(* Logix 5000 project; controller PRG_SIMON Emulate 5570 rev 30.12; software revision 30.00 *)

TASK MainTask (continuous, watchdog 5000 ms) : MainProgram

MODULES
   Local : Emulate 5570 (ICP 2, rev 30.12)
       : vendor 1 type 0 code 15 (ICP 0, rev 1.1, Output RPI 50 ms)
END_MODULES

TYPE UDT_BA :
STRUCT
   AL : BOOL[128];
END_STRUCT
END_TYPE

PROGRAM MainProgram   (* main routine MainRoutine *)
VAR
   PRG_Counter : DINT[2];
   PRG_i : DINT;
   PRG_j : DINT;
   PRG_Res_Len : DINT;
   PRG_Result : DINT[256];
   SCAN_CYCLE_TIME : DINT;
   Simon_Ciphertext : DINT[2,2];
   Simon_dec_i : DINT;
   Simon_dec_j : DINT;
   Simon_enc_i : DINT;
   Simon_enc_j : DINT;
   Simon_i : DINT;
   Simon_j : DINT;
   Simon_Plaintext : DINT[2,2];
   Simon_Rd_Max : DINT;
   Simon_Rotate_Result : DINT[2];
   Simon_Round_Keys : DINT[72,2];
   Simon_tmp1 : DINT[2];
   Simon_tmp2 : DINT[2];
   Simon_Ver : DINT;
   Simon_x : DINT[2];
   Simon_y : DINT[2];
END_VAR

ROUTINE MainRoutine   (* ladder *)
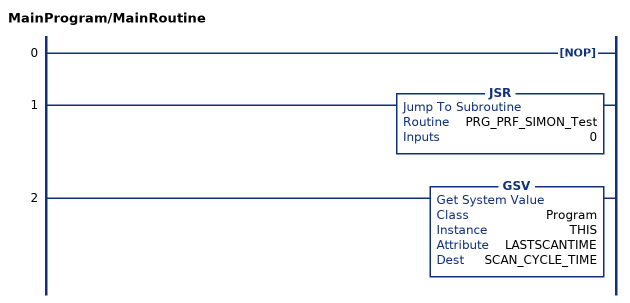
   0: NOP();
   1: JSR(PRG_PRF_SIMON_Test,0);
   2: GSV(Program,THIS,LASTSCANTIME,SCAN_CYCLE_TIME);
END_ROUTINE

ROUTINE PRG_PRF_Init   (* structured text *)
   
   
   //initialize version
   
   Simon_Ver:=2;     // 0: 32/64, 1: 64: 96, 2: 64:128, 3:128/128, 4:128/192, 5: 128/256
   
   PRG_j:=0;
   PRG_Res_Len :=  (PRG_Counter[0] AND 16#0000ffff)-1;
   
   JSR(SIMON_Init);
END_ROUTINE

ROUTINE PRG_PRF_SIMON   (* structured text *)
   // init PRG_Count[0] and PRG_Count[1] during application.. for PRF.. they could be any values
   //For PRG application, PRG_Count[0] defines the output length (i.e., the number of 64-bit, e.g., 128-bit output, PRG_Count[0]:=2)
   
   
   JSR(PRG_PRF_Init);
   PRG_j:=0;
   For PRG_i:=0 to PRG_Res_Len by 1 do
   	Simon_Plaintext[0,0]:=PRG_Counter[0]; //Upper bits of current plaintext
   	Simon_Plaintext[1,0]:=PRG_Counter[1];  //Lower bits of current plaintext
   	JSR(SIMON_Enc);
   	PRG_Result[PRG_j]:=Simon_Ciphertext[0,0];
   	PRG_Result[PRG_j+1]:=Simon_Ciphertext[1,0];
   
   	PRG_j:=PRG_j+2;
   
   End_For;
   
   JSR(SIMON_ClearKey);
   
END_ROUTINE

ROUTINE PRG_PRF_SIMON_Test   (* structured text *)
   If S:FS Then
   
   	PRG_Counter[0]:=5;
   	PRG_Counter[1]:=1;
   
   
   End_if;
   
   
   JSR(PRG_PRF_SIMON);
   
   
END_ROUTINE

ROUTINE SIMON_ClearKey   (* structured text *)
   Case Simon_Ver Of
   
   0,1,2:
   	For Simon_i:=0 to Simon_Rd_Max by 1 do
   		Simon_Round_Keys[Simon_i,0]:=0;
   	End_For;
   	Simon_tmp1[0]:=0;
   	Simon_tmp2[0]:=0;
   	Simon_Rotate_Result[0]:=0;
   3,4,5:
   	For Simon_i:=0 to Simon_Rd_Max by 1 do
   		Simon_Round_Keys[Simon_i,0]:=0;
   		Simon_Round_Keys[Simon_i,1]:=0;
   	End_For;
   	Simon_tmp1[0]:=0;
   	Simon_tmp1[1]:=0;
   	Simon_tmp2[0]:=0;
   	Simon_tmp2[1]:=0;
   	Simon_Rotate_Result[0]:=0;
   	Simon_Rotate_Result[1]:=0;
   End_Case;
   
   
END_ROUTINE

ROUTINE SIMON_Dec   (* structured text *)
   
   JSR(SIMON_Init);
   
   
   
   
   Case Simon_Ver Of
   
   0,1,2:
   	Simon_Plaintext[1,0]:=Simon_Ciphertext[0,0];
   	Simon_Plaintext[0,0]:=Simon_Ciphertext[1,0];
   
   	For Simon_i:=Simon_Rd_Max to 0 by -1 do
   		Simon_tmp2[0]:=Simon_Plaintext[0,0];  //for rotate
   		JSR(SIMON_Rotate_Left1);	//rotate based on Simon_Ciphertext[0,0]
   		Simon_tmp1[0]:= Simon_Rotate_Result[0];
   		Simon_Rotate_Result[0]:=0;
   
   		Simon_tmp2[0]:=Simon_Plaintext[0,0];  //for rotate
   		JSR(SIMON_Rotate_Left8);
   		Simon_tmp2[0]:=Simon_Rotate_Result[0];
   		Simon_tmp1[0]:= Simon_tmp1[0] AND Simon_tmp2[0];
   		Simon_Rotate_Result[0]:=0;
   
   		Simon_tmp2[0]:=Simon_Plaintext[0,0];  //for rotate
   		JSR(SIMON_Rotate_Left2);
   		Simon_tmp1[0]:= Simon_tmp1[0] XOR Simon_Rotate_Result[0];
   
   		Simon_tmp1[0]:= Simon_tmp1[0] XOR Simon_Round_Keys[Simon_i,0];
   
   		Simon_Plaintext[0,0]:= Simon_Plaintext[1,0] XOR Simon_tmp1[0];
   		Simon_Plaintext[1,0]:= Simon_tmp2[0];
   
   		Simon_Rotate_Result[0]:=0;
   
   	End_for;
   
   3,4,5:
   	Simon_Plaintext[1,0]:=Simon_Ciphertext[0,0];
   	Simon_Plaintext[1,1]:=Simon_Ciphertext[0,1];
   	Simon_Plaintext[0,0]:=Simon_Ciphertext[1,0];
   	Simon_Plaintext[0,1]:=Simon_Ciphertext[1,1];
   
   	For Simon_i:=Simon_Rd_Max to 0 by -1 do
   
   		Simon_tmp2[0]:=Simon_Plaintext[0,0];  //for rotate
   		Simon_tmp2[1]:=Simon_Plaintext[0,1];
   
   		JSR(SIMON_Rotate_Left1);	//rotate based on Simon_Ciphertext[0,0] and [0,1]
   		Simon_tmp1[0]:= Simon_Rotate_Result[0];
   		Simon_tmp1[1]:= Simon_Rotate_Result[1];
   
   		Simon_Rotate_Result[0]:=0;
   		Simon_Rotate_Result[1]:=0;
   
   		Simon_tmp2[0]:=Simon_Plaintext[0,0];
   		Simon_tmp2[1]:=Simon_Plaintext[0,1];
   		JSR(SIMON_Rotate_Left8);
   		Simon_tmp2[0]:=Simon_Rotate_Result[0];
   		Simon_tmp2[1]:=Simon_Rotate_Result[1];
   		Simon_tmp1[0]:= Simon_tmp1[0] AND Simon_tmp2[0];
   		Simon_tmp1[1]:= Simon_tmp1[1] AND Simon_tmp2[1];
   
   		Simon_tmp2[0]:=Simon_Plaintext[0,0];
   		Simon_tmp2[1]:=Simon_Plaintext[0,1];
   
   		Simon_Rotate_Result[0]:=0;
   		Simon_Rotate_Result[1]:=0;
   
   		JSR(SIMON_Rotate_Left2);
   		Simon_tmp1[0]:= Simon_tmp1[0] XOR Simon_Rotate_Result[0];
   		Simon_tmp1[1]:= Simon_tmp1[1] XOR Simon_Rotate_Result[1];
   
   		Simon_tmp1[0]:= Simon_tmp1[0] XOR Simon_Round_Keys[Simon_i,0];
   		Simon_tmp1[1]:= Simon_tmp1[1] XOR Simon_Round_Keys[Simon_i,1];
   
   
   		Simon_Plaintext[0,0]:= Simon_Plaintext[1,0] XOR Simon_tmp1[0];
   		Simon_Plaintext[0,1]:= Simon_Plaintext[1,1] XOR Simon_tmp1[1];
   
   		Simon_Plaintext[1,0]:= Simon_tmp2[0];
   		Simon_Plaintext[1,1]:= Simon_tmp2[1];
   
   		Simon_Rotate_Result[0]:=0;
   		Simon_Rotate_Result[1]:=0;
   
   	End_for;
   
   End_Case;
   
   
   
   
   
   
   JSR(SIMON_ClearKey);
   
   
   
   
   
   
   
   
END_ROUTINE

ROUTINE SIMON_Enc   (* structured text *)
   
   Case Simon_Ver Of
   
   0,1,2:
   	//Simon_Ciphertext[1,0]:=Simon_Plaintext[0,0];
   	//Simon_Ciphertext[0,0]:=Simon_Plaintext[1,0];
   
   	Simon_Ciphertext[0,0]:=Simon_Plaintext[1,0];
   	Simon_Ciphertext[1,0]:=Simon_Plaintext[0,0];
   
   	For Simon_i:=0 to Simon_Rd_Max by 1 do
   		Simon_tmp2[0]:=Simon_Ciphertext[0,0];  //for rotate
   		JSR(SIMON_Rotate_Left1);	//rotate based on Simon_Plaintext[0,0]
   		Simon_tmp1[0]:= Simon_Rotate_Result[0];
   		Simon_Rotate_Result[0]:=0;
   
   		Simon_tmp2[0]:=Simon_Ciphertext[0,0];  //for rotate
   		JSR(SIMON_Rotate_Left8);
   		Simon_tmp2[0]:=Simon_Rotate_Result[0];
   
   		Simon_tmp1[0]:= Simon_tmp1[0] AND Simon_tmp2[0];
   		Simon_Rotate_Result[0]:=0;
   
   		Simon_tmp2[0]:=Simon_Ciphertext[0,0];  //for rotate
   		JSR(SIMON_Rotate_Left2);
   		Simon_tmp1[0]:= Simon_tmp1[0] XOR Simon_Rotate_Result[0];
   
   		Simon_tmp1[0]:= Simon_tmp1[0] XOR Simon_Round_Keys[Simon_i,0];
   
   		Simon_Ciphertext[0,0]:= Simon_Ciphertext[1,0] XOR Simon_tmp1[0];
   		Simon_Ciphertext[1,0]:= Simon_tmp2[0];
   
   		Simon_Rotate_Result[0]:=0;
   
   	End_for;
   
   3,4,5:
   	Simon_Ciphertext[1,0]:=Simon_Plaintext[0,0];
   	Simon_Ciphertext[1,1]:=Simon_Plaintext[0,1];
   	Simon_Ciphertext[0,0]:=Simon_Plaintext[1,0];
   	Simon_Ciphertext[0,1]:=Simon_Plaintext[1,1];
   
   	For Simon_i:=0 to Simon_Rd_Max by 1 do
   
   		Simon_tmp2[0]:=Simon_Ciphertext[0,0];  //for rotate
   		Simon_tmp2[1]:=Simon_Ciphertext[0,1];
   
   		JSR(SIMON_Rotate_Left1);	//rotate based on Simon_Plaintext[0,0] and [0,1]
   		Simon_tmp1[0]:= Simon_Rotate_Result[0];
   		Simon_tmp1[1]:= Simon_Rotate_Result[1];
   
   		Simon_Rotate_Result[0]:=0;
   		Simon_Rotate_Result[1]:=0;
   
   		Simon_tmp2[0]:=Simon_Ciphertext[0,0];
   		Simon_tmp2[1]:=Simon_Ciphertext[0,1];
   		JSR(SIMON_Rotate_Left8);
   		Simon_tmp2[0]:=Simon_Rotate_Result[0];
   		Simon_tmp2[1]:=Simon_Rotate_Result[1];
   		Simon_tmp1[0]:= Simon_tmp1[0] AND Simon_tmp2[0];
   		Simon_tmp1[1]:= Simon_tmp1[1] AND Simon_tmp2[1];
   
   		Simon_Rotate_Result[0]:=0;
   		Simon_Rotate_Result[1]:=0;
   
   		Simon_tmp2[0]:=Simon_Ciphertext[0,0];
   		Simon_tmp2[1]:=Simon_Ciphertext[0,1];
   		JSR(SIMON_Rotate_Left2);
   		Simon_tmp1[0]:= Simon_tmp1[0] XOR Simon_Rotate_Result[0];
   		Simon_tmp1[1]:= Simon_tmp1[1] XOR Simon_Rotate_Result[1];
   
   		Simon_tmp1[0]:= Simon_tmp1[0] XOR Simon_Round_Keys[Simon_i,0];
   		Simon_tmp1[1]:= Simon_tmp1[1] XOR Simon_Round_Keys[Simon_i,1];
   
   
   		Simon_Ciphertext[0,0]:= Simon_Ciphertext[1,0] XOR Simon_tmp1[0];
   		Simon_Ciphertext[0,1]:= Simon_Ciphertext[1,1] XOR Simon_tmp1[1];
   
   		Simon_Ciphertext[1,0]:= Simon_tmp2[0];
   		Simon_Ciphertext[1,1]:= Simon_tmp2[1];
   
   		Simon_Rotate_Result[0]:=0;
   		Simon_Rotate_Result[1]:=0;
   
   	End_for;
   
   End_Case;
   
   
   
   
   
   JSR(SIMON_ClearKey);
   
   
   
   
   
   
END_ROUTINE

ROUTINE SIMON_Init   (* structured text *)
   CASE Simon_Ver Of
   	0:
   		Simon_Rd_Max:=31;
   		Simon_Round_Keys[0,0]:=58892;
   		Simon_Round_Keys[1,0]:=17469;
   		Simon_Round_Keys[2,0]:=46338;
   		Simon_Round_Keys[3,0]:=24531;
   		Simon_Round_Keys[4,0]:=28834;
   		Simon_Round_Keys[5,0]:=46808;
   		Simon_Round_Keys[6,0]:=58663;
   		Simon_Round_Keys[7,0]:=25382;
   		Simon_Round_Keys[8,0]:=44074;
   		Simon_Round_Keys[9,0]:=20080;
   		Simon_Round_Keys[10,0]:=29824;
   		Simon_Round_Keys[11,0]:=27762;
   		Simon_Round_Keys[12,0]:=59835;
   		Simon_Round_Keys[13,0]:=7335;
   		Simon_Round_Keys[14,0]:=61675;
   		Simon_Round_Keys[15,0]:=21004;
   		Simon_Round_Keys[16,0]:=30396;
   		Simon_Round_Keys[17,0]:=49986;
   		Simon_Round_Keys[18,0]:=30611;
   		Simon_Round_Keys[19,0]:=24687;
   		Simon_Round_Keys[20,0]:=51228;
   		Simon_Round_Keys[21,0]:=43363;
   		Simon_Round_Keys[22,0]:=53306;
   		Simon_Round_Keys[23,0]:=31273;
   		Simon_Round_Keys[24,0]:=32558;
   		Simon_Round_Keys[25,0]:=3536;
   		Simon_Round_Keys[26,0]:=26948;
   		Simon_Round_Keys[27,0]:=48822;
   		Simon_Round_Keys[28,0]:=19540;
   		Simon_Round_Keys[29,0]:=7940;
   		Simon_Round_Keys[30,0]:=35612;
   		Simon_Round_Keys[31,0]:=30709;
   	1:
   		Simon_Rd_Max:=41;
   		Simon_Round_Keys[0,0]:=797923611;
   		Simon_Round_Keys[1,0]:=1435100883;
   		Simon_Round_Keys[2,0]:=570050683;
   		Simon_Round_Keys[3,0]:=1467839184;
   		Simon_Round_Keys[4,0]:=862930168;
   		Simon_Round_Keys[5,0]:=1472127870;
   		Simon_Round_Keys[6,0]:=-834641963;
   		Simon_Round_Keys[7,0]:=1294397471;
   		Simon_Round_Keys[8,0]:=923082899;
   		Simon_Round_Keys[9,0]:=-1414689665;
   		Simon_Round_Keys[10,0]:=292004807;
   		Simon_Round_Keys[11,0]:=1508575081;
   		Simon_Round_Keys[12,0]:=-203282145;
   		Simon_Round_Keys[13,0]:=-1842036876;
   		Simon_Round_Keys[14,0]:=1503726394;
   		Simon_Round_Keys[15,0]:=1138111690;
   		Simon_Round_Keys[16,0]:=213599617;
   		Simon_Round_Keys[17,0]:=1619530791;
   		Simon_Round_Keys[18,0]:=1385821355;
   		Simon_Round_Keys[19,0]:=-1593573967;
   		Simon_Round_Keys[20,0]:=-1780152310;
   		Simon_Round_Keys[21,0]:=-1546357816;
   		Simon_Round_Keys[22,0]:=1899435;
   		Simon_Round_Keys[23,0]:=1461836050;
   		Simon_Round_Keys[24,0]:=-2061126966;
   		Simon_Round_Keys[25,0]:=1732697272;
   		Simon_Round_Keys[26,0]:=1817790448;
   		Simon_Round_Keys[27,0]:=-785825972;
   		Simon_Round_Keys[28,0]:=-987783455;
   		Simon_Round_Keys[29,0]:=186588167;
   		Simon_Round_Keys[30,0]:=-1367749570;
   		Simon_Round_Keys[31,0]:=-1535518601;
   		Simon_Round_Keys[32,0]:=241059013;
   		Simon_Round_Keys[33,0]:=-708545457;
   		Simon_Round_Keys[34,0]:=-514880440;
   		Simon_Round_Keys[35,0]:=1351987569;
   		Simon_Round_Keys[36,0]:=-140601681;
   		Simon_Round_Keys[37,0]:=784661324;
   		Simon_Round_Keys[38,0]:=-1947799209;
   		Simon_Round_Keys[39,0]:=-1872190481;
   		Simon_Round_Keys[40,0]:=-1911353564;
   		Simon_Round_Keys[41,0]:=-985279030;
   	2:
   		Simon_Rd_Max:=43;
   		Simon_Round_Keys[0,0]:=-1252640063;
   		Simon_Round_Keys[1,0]:=16063003;
   		Simon_Round_Keys[2,0]:=-1716801011;
   		Simon_Round_Keys[3,0]:=294058422;
   		Simon_Round_Keys[4,0]:=-2089218819;
   		Simon_Round_Keys[5,0]:=-1093170128;
   		Simon_Round_Keys[6,0]:=-1408927769;
   		Simon_Round_Keys[7,0]:=1282112963;
   		Simon_Round_Keys[8,0]:=1509852702;
   		Simon_Round_Keys[9,0]:=-367591186;
   		Simon_Round_Keys[10,0]:=-313151875;
   		Simon_Round_Keys[11,0]:=2026360408;
   		Simon_Round_Keys[12,0]:=1690726407;
   		Simon_Round_Keys[13,0]:=-145773523;
   		Simon_Round_Keys[14,0]:=-1945611938;
   		Simon_Round_Keys[15,0]:=-219020842;
   		Simon_Round_Keys[16,0]:=-347126000;
   		Simon_Round_Keys[17,0]:=-958819553;
   		Simon_Round_Keys[18,0]:=-1914268711;
   		Simon_Round_Keys[19,0]:=-740974030;
   		Simon_Round_Keys[20,0]:=622799657;
   		Simon_Round_Keys[21,0]:=846511031;
   		Simon_Round_Keys[22,0]:=770436402;
   		Simon_Round_Keys[23,0]:=1064131354;
   		Simon_Round_Keys[24,0]:=-979770697;
   		Simon_Round_Keys[25,0]:=-1460359263;
   		Simon_Round_Keys[26,0]:=-248461252;
   		Simon_Round_Keys[27,0]:=-1885850817;
   		Simon_Round_Keys[28,0]:=-1448880025;
   		Simon_Round_Keys[29,0]:=-334653330;
   		Simon_Round_Keys[30,0]:=-1695993890;
   		Simon_Round_Keys[31,0]:=205839422;
   		Simon_Round_Keys[32,0]:=1047207403;
   		Simon_Round_Keys[33,0]:=-1688236183;
   		Simon_Round_Keys[34,0]:=-1646939783;
   		Simon_Round_Keys[35,0]:=-395364148;
   		Simon_Round_Keys[36,0]:=-1723851930;
   		Simon_Round_Keys[37,0]:=-1144586697;
   		Simon_Round_Keys[38,0]:=1973127706;
   		Simon_Round_Keys[39,0]:=1218994850;
   		Simon_Round_Keys[40,0]:=-1658111848;
   		Simon_Round_Keys[41,0]:=471575198;
   		Simon_Round_Keys[42,0]:=-1139438973;
   		Simon_Round_Keys[43,0]:=-1377481455;
   	3:
   		Simon_Rd_Max:=67;
   		Simon_Round_Keys[0,0]:=-907025205;
   		Simon_Round_Keys[0,1]:=207142458;
   		Simon_Round_Keys[1,0]:=-652646316;
   		Simon_Round_Keys[1,1]:=252011832;
   		Simon_Round_Keys[2,0]:=1958888637;
   		Simon_Round_Keys[2,1]:=-256542565;
   		Simon_Round_Keys[3,0]:=1016210364;
   		Simon_Round_Keys[3,1]:=1561640341;
   		Simon_Round_Keys[4,0]:=-2044158199;
   		Simon_Round_Keys[4,1]:=-951092617;
   		Simon_Round_Keys[5,0]:=857846596;
   		Simon_Round_Keys[5,1]:=-2974950;
   		Simon_Round_Keys[6,0]:=-340233113;
   		Simon_Round_Keys[6,1]:=1631310078;
   		Simon_Round_Keys[7,0]:=-1058274422;
   		Simon_Round_Keys[7,1]:=1411361121;
   		Simon_Round_Keys[8,0]:=1630436302;
   		Simon_Round_Keys[8,1]:=1310593161;
   		Simon_Round_Keys[9,0]:=-2083539204;
   		Simon_Round_Keys[9,1]:=-600138873;
   		Simon_Round_Keys[10,0]:=2004212402;
   		Simon_Round_Keys[10,1]:=-1161434199;
   		Simon_Round_Keys[11,0]:=-1295502075;
   		Simon_Round_Keys[11,1]:=-1836927347;
   		Simon_Round_Keys[12,0]:=419739346;
   		Simon_Round_Keys[12,1]:=336580700;
   		Simon_Round_Keys[13,0]:=407780687;
   		Simon_Round_Keys[13,1]:=1907925923;
   		Simon_Round_Keys[14,0]:=-1521151868;
   		Simon_Round_Keys[14,1]:=1977604119;
   		Simon_Round_Keys[15,0]:=896154083;
   		Simon_Round_Keys[15,1]:=1466082827;
   		Simon_Round_Keys[16,0]:=1558686575;
   		Simon_Round_Keys[16,1]:=862239939;
   		Simon_Round_Keys[17,0]:=114071154;
   		Simon_Round_Keys[17,1]:=-1871601199;
   		Simon_Round_Keys[18,0]:=-607890295;
   		Simon_Round_Keys[18,1]:=1299568338;
   		Simon_Round_Keys[19,0]:=1045657693;
   		Simon_Round_Keys[19,1]:=-161177025;
   		Simon_Round_Keys[20,0]:=-688480272;
   		Simon_Round_Keys[20,1]:=1084529385;
   		Simon_Round_Keys[21,0]:=-357674769;
   		Simon_Round_Keys[21,1]:=479541203;
   		Simon_Round_Keys[22,0]:=886380795;
   		Simon_Round_Keys[22,1]:=43094520;
   		Simon_Round_Keys[23,0]:=1044809980;
   		Simon_Round_Keys[23,1]:=281979091;
   		Simon_Round_Keys[24,0]:=1873480662;
   		Simon_Round_Keys[24,1]:=-487618466;
   		Simon_Round_Keys[25,0]:=1980441222;
   		Simon_Round_Keys[25,1]:=130356366;
   		Simon_Round_Keys[26,0]:=147290141;
   		Simon_Round_Keys[26,1]:=1001239497;
   		Simon_Round_Keys[27,0]:=303043151;
   		Simon_Round_Keys[27,1]:=1647097004;
   		Simon_Round_Keys[28,0]:=1807345483;
   		Simon_Round_Keys[28,1]:=279873862;
   		Simon_Round_Keys[29,0]:=624398167;
   		Simon_Round_Keys[29,1]:=-1930256593;
   		Simon_Round_Keys[30,0]:=-1865894730;
   		Simon_Round_Keys[30,1]:=139359338;
   		Simon_Round_Keys[31,0]:=-789874473;
   		Simon_Round_Keys[31,1]:=-688307584;
   		Simon_Round_Keys[32,0]:=-31833823;
   		Simon_Round_Keys[32,1]:=2118832481;
   		Simon_Round_Keys[33,0]:=-1739557682;
   		Simon_Round_Keys[33,1]:=425587835;
   		Simon_Round_Keys[34,0]:=1747895794;
   		Simon_Round_Keys[34,1]:=319052991;
   		Simon_Round_Keys[35,0]:=846789164;
   		Simon_Round_Keys[35,1]:=-81285290;
   		Simon_Round_Keys[36,0]:=938446948;
   		Simon_Round_Keys[36,1]:=2109714568;
   		Simon_Round_Keys[37,0]:=-739547817;
   		Simon_Round_Keys[37,1]:=1398480993;
   		Simon_Round_Keys[38,0]:=1544595246;
   		Simon_Round_Keys[38,1]:=126637793;
   		Simon_Round_Keys[39,0]:=860925059;
   		Simon_Round_Keys[39,1]:=1448543639;
   		Simon_Round_Keys[40,0]:=2143392852;
   		Simon_Round_Keys[40,1]:=-716656265;
   		Simon_Round_Keys[41,0]:=-1372939347;
   		Simon_Round_Keys[41,1]:=-435344985;
   		Simon_Round_Keys[42,0]:=-567769089;
   		Simon_Round_Keys[42,1]:=2068633297;
   		Simon_Round_Keys[43,0]:=-1350526428;
   		Simon_Round_Keys[43,1]:=-1036555675;
   		Simon_Round_Keys[44,0]:=1947003070;
   		Simon_Round_Keys[44,1]:=1115220787;
   		Simon_Round_Keys[45,0]:=1719425706;
   		Simon_Round_Keys[45,1]:=-900359920;
   		Simon_Round_Keys[46,0]:=-192002717;
   		Simon_Round_Keys[46,1]:=-1080759493;
   		Simon_Round_Keys[47,0]:=-812345260;
   		Simon_Round_Keys[47,1]:=1248711085;
   		Simon_Round_Keys[48,0]:=-1046160164;
   		Simon_Round_Keys[48,1]:=-1044799936;
   		Simon_Round_Keys[49,0]:=924943140;
   		Simon_Round_Keys[49,1]:=2123163808;
   		Simon_Round_Keys[50,0]:=2039689938;
   		Simon_Round_Keys[50,1]:=1669705323;
   		Simon_Round_Keys[51,0]:=2090908127;
   		Simon_Round_Keys[51,1]:=-765821324;
   		Simon_Round_Keys[52,0]:=2116873771;
   		Simon_Round_Keys[52,1]:=2076462446;
   		Simon_Round_Keys[53,0]:=1652656677;
   		Simon_Round_Keys[53,1]:=-710090652;
   		Simon_Round_Keys[54,0]:=747712652;
   		Simon_Round_Keys[54,1]:=-839007496;
   		Simon_Round_Keys[55,0]:=1498717196;
   		Simon_Round_Keys[55,1]:=-1998348751;
   		Simon_Round_Keys[56,0]:=1217062049;
   		Simon_Round_Keys[56,1]:=30319515;
   		Simon_Round_Keys[57,0]:=-968613802;
   		Simon_Round_Keys[57,1]:=69894377;
   		Simon_Round_Keys[58,0]:=-1120694706;
   		Simon_Round_Keys[58,1]:=845480917;
   		Simon_Round_Keys[59,0]:=-604585981;
   		Simon_Round_Keys[59,1]:=1958413752;
   		Simon_Round_Keys[60,0]:=-939405585;
   		Simon_Round_Keys[60,1]:=-810171409;
   		Simon_Round_Keys[61,0]:=1288373833;
   		Simon_Round_Keys[61,1]:=-1623024215;
   		Simon_Round_Keys[62,0]:=-352925090;
   		Simon_Round_Keys[62,1]:=-1422629559;
   		Simon_Round_Keys[63,0]:=204320471;
   		Simon_Round_Keys[63,1]:=690314999;
   		Simon_Round_Keys[64,0]:=545914512;
   		Simon_Round_Keys[64,1]:=1957631435;
   		Simon_Round_Keys[65,0]:=-1823377808;
   		Simon_Round_Keys[65,1]:=592748548;
   		Simon_Round_Keys[66,0]:=-27602894;
   		Simon_Round_Keys[66,1]:=-1165333650;
   		Simon_Round_Keys[67,0]:=-29434619;
   		Simon_Round_Keys[67,1]:=116469945;
   	4:
   		Simon_Rd_Max:=68;
   		Simon_Round_Keys[0,0]:=1027963089;
   		Simon_Round_Keys[0,1]:=544430627;
   		Simon_Round_Keys[1,0]:=-683055369;
   		Simon_Round_Keys[1,1]:=37620279;
   		Simon_Round_Keys[2,0]:=534363766;
   		Simon_Round_Keys[2,1]:=1064974017;
   		Simon_Round_Keys[3,0]:=923873478;
   		Simon_Round_Keys[3,1]:=270623091;
   		Simon_Round_Keys[4,0]:=982158941;
   		Simon_Round_Keys[4,1]:=1019254631;
   		Simon_Round_Keys[5,0]:=-1110644030;
   		Simon_Round_Keys[5,1]:=-960660674;
   		Simon_Round_Keys[6,0]:=-1538144672;
   		Simon_Round_Keys[6,1]:=1455331749;
   		Simon_Round_Keys[7,0]:=1989098669;
   		Simon_Round_Keys[7,1]:=430058512;
   		Simon_Round_Keys[8,0]:=1078593005;
   		Simon_Round_Keys[8,1]:=-1724677879;
   		Simon_Round_Keys[9,0]:=-278389100;
   		Simon_Round_Keys[9,1]:=-1678163493;
   		Simon_Round_Keys[10,0]:=2025995703;
   		Simon_Round_Keys[10,1]:=-848393262;
   		Simon_Round_Keys[11,0]:=506793134;
   		Simon_Round_Keys[11,1]:=-1094895774;
   		Simon_Round_Keys[12,0]:=-798127997;
   		Simon_Round_Keys[12,1]:=1743653272;
   		Simon_Round_Keys[13,0]:=1371401022;
   		Simon_Round_Keys[13,1]:=-1206429906;
   		Simon_Round_Keys[14,0]:=953785041;
   		Simon_Round_Keys[14,1]:=-1366647699;
   		Simon_Round_Keys[15,0]:=1683788482;
   		Simon_Round_Keys[15,1]:=692595039;
   		Simon_Round_Keys[16,0]:=1020324615;
   		Simon_Round_Keys[16,1]:=-743107565;
   		Simon_Round_Keys[17,0]:=-1004392916;
   		Simon_Round_Keys[17,1]:=-1274670986;
   		Simon_Round_Keys[18,0]:=1575449145;
   		Simon_Round_Keys[18,1]:=255278374;
   		Simon_Round_Keys[19,0]:=-767761648;
   		Simon_Round_Keys[19,1]:=371737674;
   		Simon_Round_Keys[20,0]:=1737719541;
   		Simon_Round_Keys[20,1]:=-715714489;
   		Simon_Round_Keys[21,0]:=-416550399;
   		Simon_Round_Keys[21,1]:=2023442159;
   		Simon_Round_Keys[22,0]:=1010988410;
   		Simon_Round_Keys[22,1]:=1607727896;
   		Simon_Round_Keys[23,0]:=-42418452;
   		Simon_Round_Keys[23,1]:=2125915837;
   		Simon_Round_Keys[24,0]:=1951441604;
   		Simon_Round_Keys[24,1]:=-1623465908;
   		Simon_Round_Keys[25,0]:=-7386454;
   		Simon_Round_Keys[25,1]:=-1328690690;
   		Simon_Round_Keys[26,0]:=-1344033323;
   		Simon_Round_Keys[26,1]:=-1030851353;
   		Simon_Round_Keys[27,0]:=257115250;
   		Simon_Round_Keys[27,1]:=-2054285712;
   		Simon_Round_Keys[28,0]:=-682199050;
   		Simon_Round_Keys[28,1]:=379885290;
   		Simon_Round_Keys[29,0]:=824441886;
   		Simon_Round_Keys[29,1]:=161376620;
   		Simon_Round_Keys[30,0]:=662829832;
   		Simon_Round_Keys[30,1]:=-1741304273;
   		Simon_Round_Keys[31,0]:=713196507;
   		Simon_Round_Keys[31,1]:=-922649281;
   		Simon_Round_Keys[32,0]:=-207271469;
   		Simon_Round_Keys[32,1]:=-756494328;
   		Simon_Round_Keys[33,0]:=-842193338;
   		Simon_Round_Keys[33,1]:=1437520944;
   		Simon_Round_Keys[34,0]:=-2073912023;
   		Simon_Round_Keys[34,1]:=200548852;
   		Simon_Round_Keys[35,0]:=-1463508582;
   		Simon_Round_Keys[35,1]:=-572374223;
   		Simon_Round_Keys[36,0]:=203314750;
   		Simon_Round_Keys[36,1]:=-587113789;
   		Simon_Round_Keys[37,0]:=1776200792;
   		Simon_Round_Keys[37,1]:=-1640544322;
   		Simon_Round_Keys[38,0]:=472046693;
   		Simon_Round_Keys[38,1]:=422499107;
   		Simon_Round_Keys[39,0]:=610635530;
   		Simon_Round_Keys[39,1]:=1061707223;
   		Simon_Round_Keys[40,0]:=-1778624947;
   		Simon_Round_Keys[40,1]:=-484558810;
   		Simon_Round_Keys[41,0]:=287093996;
   		Simon_Round_Keys[41,1]:=-601824417;
   		Simon_Round_Keys[42,0]:=1790710963;
   		Simon_Round_Keys[42,1]:=1523696625;
   		Simon_Round_Keys[43,0]:=930473490;
   		Simon_Round_Keys[43,1]:=-1912972041;
   		Simon_Round_Keys[44,0]:=-2092080210;
   		Simon_Round_Keys[44,1]:=-1815607971;
   		Simon_Round_Keys[45,0]:=-1020146586;
   		Simon_Round_Keys[45,1]:=-1633114229;
   		Simon_Round_Keys[46,0]:=-802509128;
   		Simon_Round_Keys[46,1]:=-979886508;
   		Simon_Round_Keys[47,0]:=-198112412;
   		Simon_Round_Keys[47,1]:=950077700;
   		Simon_Round_Keys[48,0]:=1164940256;
   		Simon_Round_Keys[48,1]:=1897890474;
   		Simon_Round_Keys[49,0]:=581792523;
   		Simon_Round_Keys[49,1]:=-1946127422;
   		Simon_Round_Keys[50,0]:=-1555808995;
   		Simon_Round_Keys[50,1]:=-1170768221;
   		Simon_Round_Keys[51,0]:=1131325910;
   		Simon_Round_Keys[51,1]:=-951040834;
   		Simon_Round_Keys[52,0]:=1301525596;
   		Simon_Round_Keys[52,1]:=-533749829;
   		Simon_Round_Keys[53,0]:=-217336772;
   		Simon_Round_Keys[53,1]:=-1184623097;
   		Simon_Round_Keys[54,0]:=-1461546436;
   		Simon_Round_Keys[54,1]:=-636736463;
   		Simon_Round_Keys[55,0]:=-1341741310;
   		Simon_Round_Keys[55,1]:=-1903848935;
   		Simon_Round_Keys[56,0]:=151294612;
   		Simon_Round_Keys[56,1]:=1095010263;
   		Simon_Round_Keys[57,0]:=-1678471265;
   		Simon_Round_Keys[57,1]:=1091008408;
   		Simon_Round_Keys[58,0]:=-895810787;
   		Simon_Round_Keys[58,1]:=1716123676;
   		Simon_Round_Keys[59,0]:=-1884278352;
   		Simon_Round_Keys[59,1]:=1472181849;
   		Simon_Round_Keys[60,0]:=1232945823;
   		Simon_Round_Keys[60,1]:=-845315976;
   		Simon_Round_Keys[61,0]:=-2024172149;
   		Simon_Round_Keys[61,1]:=-1006271118;
   		Simon_Round_Keys[62,0]:=-1134131484;
   		Simon_Round_Keys[62,1]:=-251728537;
   		Simon_Round_Keys[63,0]:=-41830285;
   		Simon_Round_Keys[63,1]:=705798069;
   		Simon_Round_Keys[64,0]:=1907567858;
   		Simon_Round_Keys[64,1]:=492968773;
   		Simon_Round_Keys[65,0]:=226226000;
   		Simon_Round_Keys[65,1]:=546967460;
   		Simon_Round_Keys[66,0]:=146725525;
   		Simon_Round_Keys[66,1]:=1755871824;
   		Simon_Round_Keys[67,0]:=-1578952937;
   		Simon_Round_Keys[67,1]:=414174385;
   		Simon_Round_Keys[68,0]:=-567597680;
   		Simon_Round_Keys[68,1]:=-1101092678;
   	5:
   		Simon_Rd_Max:=71;
   		Simon_Round_Keys[0,0]:=-390970254;
   		Simon_Round_Keys[0,1]:=1985106510;
   		Simon_Round_Keys[1,0]:=836986459;
   		Simon_Round_Keys[1,1]:=-830713793;
   		Simon_Round_Keys[2,0]:=978164418;
   		Simon_Round_Keys[2,1]:=-1961661141;
   		Simon_Round_Keys[3,0]:=765693446;
   		Simon_Round_Keys[3,1]:=-1200877126;
   		Simon_Round_Keys[4,0]:=1837819274;
   		Simon_Round_Keys[4,1]:=-1324964684;
   		Simon_Round_Keys[5,0]:=-168663280;
   		Simon_Round_Keys[5,1]:=-1757183886;
   		Simon_Round_Keys[6,0]:=1579613877;
   		Simon_Round_Keys[6,1]:=-1027206398;
   		Simon_Round_Keys[7,0]:=989787679;
   		Simon_Round_Keys[7,1]:=-9335540;
   		Simon_Round_Keys[8,0]:=-425887052;
   		Simon_Round_Keys[8,1]:=1407000841;
   		Simon_Round_Keys[9,0]:=-318642983;
   		Simon_Round_Keys[9,1]:=-673261925;
   		Simon_Round_Keys[10,0]:=791642980;
   		Simon_Round_Keys[10,1]:=-1496664303;
   		Simon_Round_Keys[11,0]:=-1441334785;
   		Simon_Round_Keys[11,1]:=627071168;
   		Simon_Round_Keys[12,0]:=749592252;
   		Simon_Round_Keys[12,1]:=-2125721768;
   		Simon_Round_Keys[13,0]:=1138494870;
   		Simon_Round_Keys[13,1]:=-779258978;
   		Simon_Round_Keys[14,0]:=-2102417481;
   		Simon_Round_Keys[14,1]:=-778157648;
   		Simon_Round_Keys[15,0]:=915263195;
   		Simon_Round_Keys[15,1]:=-1208216313;
   		Simon_Round_Keys[16,0]:=-1619685782;
   		Simon_Round_Keys[16,1]:=1530783530;
   		Simon_Round_Keys[17,0]:=894219664;
   		Simon_Round_Keys[17,1]:=927689220;
   		Simon_Round_Keys[18,0]:=727657132;
   		Simon_Round_Keys[18,1]:=-1086505095;
   		Simon_Round_Keys[19,0]:=-1606623160;
   		Simon_Round_Keys[19,1]:=1472430846;
   		Simon_Round_Keys[20,0]:=2060946409;
   		Simon_Round_Keys[20,1]:=187092954;
   		Simon_Round_Keys[21,0]:=-1982133367;
   		Simon_Round_Keys[21,1]:=-1708158977;
   		Simon_Round_Keys[22,0]:=-116564438;
   		Simon_Round_Keys[22,1]:=1431713434;
   		Simon_Round_Keys[23,0]:=-531961211;
   		Simon_Round_Keys[23,1]:=1350042290;
   		Simon_Round_Keys[24,0]:=1534294247;
   		Simon_Round_Keys[24,1]:=-434018864;
   		Simon_Round_Keys[25,0]:=1674179828;
   		Simon_Round_Keys[25,1]:=1487719310;
   		Simon_Round_Keys[26,0]:=1735400901;
   		Simon_Round_Keys[26,1]:=444333297;
   		Simon_Round_Keys[27,0]:=799581701;
   		Simon_Round_Keys[27,1]:=1143488433;
   		Simon_Round_Keys[28,0]:=-979537010;
   		Simon_Round_Keys[28,1]:=1819648252;
   		Simon_Round_Keys[29,0]:=-1606864701;
   		Simon_Round_Keys[29,1]:=-97346557;
   		Simon_Round_Keys[30,0]:=1441248171;
   		Simon_Round_Keys[30,1]:=-375742643;
   		Simon_Round_Keys[31,0]:=81745149;
   		Simon_Round_Keys[31,1]:=-1665556590;
   		Simon_Round_Keys[32,0]:=157402215;
   		Simon_Round_Keys[32,1]:=-1337369234;
   		Simon_Round_Keys[33,0]:=533148948;
   		Simon_Round_Keys[33,1]:=-1444102471;
   		Simon_Round_Keys[34,0]:=-54028912;
   		Simon_Round_Keys[34,1]:=1295386257;
   		Simon_Round_Keys[35,0]:=-1852675451;
   		Simon_Round_Keys[35,1]:=1979939964;
   		Simon_Round_Keys[36,0]:=1933481617;
   		Simon_Round_Keys[36,1]:=276746073;
   		Simon_Round_Keys[37,0]:=248732650;
   		Simon_Round_Keys[37,1]:=-379002890;
   		Simon_Round_Keys[38,0]:=2037897468;
   		Simon_Round_Keys[38,1]:=-1661166802;
   		Simon_Round_Keys[39,0]:=-104405666;
   		Simon_Round_Keys[39,1]:=2129801934;
   		Simon_Round_Keys[40,0]:=334654544;
   		Simon_Round_Keys[40,1]:=1371228092;
   		Simon_Round_Keys[41,0]:=-1128005728;
   		Simon_Round_Keys[41,1]:=-1058012097;
   		Simon_Round_Keys[42,0]:=907395048;
   		Simon_Round_Keys[42,1]:=341199413;
   		Simon_Round_Keys[43,0]:=-548089632;
   		Simon_Round_Keys[43,1]:=-1138225551;
   		Simon_Round_Keys[44,0]:=1894221806;
   		Simon_Round_Keys[44,1]:=-2118911188;
   		Simon_Round_Keys[45,0]:=-363847261;
   		Simon_Round_Keys[45,1]:=-1190918910;
   		Simon_Round_Keys[46,0]:=-440509844;
   		Simon_Round_Keys[46,1]:=-382825287;
   		Simon_Round_Keys[47,0]:=-1434378233;
   		Simon_Round_Keys[47,1]:=-1163710374;
   		Simon_Round_Keys[48,0]:=1296053343;
   		Simon_Round_Keys[48,1]:=-1290583990;
   		Simon_Round_Keys[49,0]:=-690486976;
   		Simon_Round_Keys[49,1]:=80317725;
   		Simon_Round_Keys[50,0]:=741085871;
   		Simon_Round_Keys[50,1]:=-848507050;
   		Simon_Round_Keys[51,0]:=1059717164;
   		Simon_Round_Keys[51,1]:=-1678026070;
   		Simon_Round_Keys[52,0]:=-1991274156;
   		Simon_Round_Keys[52,1]:=-439382912;
   		Simon_Round_Keys[53,0]:=-406584208;
   		Simon_Round_Keys[53,1]:=-1935425251;
   		Simon_Round_Keys[54,0]:=452750798;
   		Simon_Round_Keys[54,1]:=-1142475824;
   		Simon_Round_Keys[55,0]:=-1800712837;
   		Simon_Round_Keys[55,1]:=-2073917552;
   		Simon_Round_Keys[56,0]:=-371577847;
   		Simon_Round_Keys[56,1]:=-1858573134;
   		Simon_Round_Keys[57,0]:=828962943;
   		Simon_Round_Keys[57,1]:=-2135315397;
   		Simon_Round_Keys[58,0]:=251653042;
   		Simon_Round_Keys[58,1]:=1276049708;
   		Simon_Round_Keys[59,0]:=-2103327965;
   		Simon_Round_Keys[59,1]:=-465361183;
   		Simon_Round_Keys[60,0]:=-752089612;
   		Simon_Round_Keys[60,1]:=-422955194;
   		Simon_Round_Keys[61,0]:=592073186;
   		Simon_Round_Keys[61,1]:=-1965539393;
   		Simon_Round_Keys[62,0]:=718147157;
   		Simon_Round_Keys[62,1]:=933460194;
   		Simon_Round_Keys[63,0]:=-105342454;
   		Simon_Round_Keys[63,1]:=-441681408;
   		Simon_Round_Keys[64,0]:=-1588818950;
   		Simon_Round_Keys[64,1]:=-1581490158;
   		Simon_Round_Keys[65,0]:=-1047262546;
   		Simon_Round_Keys[65,1]:=1696023995;
   		Simon_Round_Keys[66,0]:=211260518;
   		Simon_Round_Keys[66,1]:=-1698176700;
   		Simon_Round_Keys[67,0]:=-2007464224;
   		Simon_Round_Keys[67,1]:=1508453628;
   		Simon_Round_Keys[68,0]:=-833914798;
   		Simon_Round_Keys[68,1]:=172159094;
   		Simon_Round_Keys[69,0]:=749838461;
   		Simon_Round_Keys[69,1]:=-1426543072;
   		Simon_Round_Keys[70,0]:=-2010462636;
   		Simon_Round_Keys[70,1]:=-873339522;
   		Simon_Round_Keys[71,0]:=-217169763;
   		Simon_Round_Keys[71,1]:=-754881756;
   End_CASE;
   
END_ROUTINE

ROUTINE SIMON_Rotate_Left1   (* structured text *)
   CASE Simon_Ver Of
   	0:
   		Simon_Rotate_Result[0].[0]:=Simon_tmp2[0].[15];
   		Simon_Rotate_Result[0].[15]:=Simon_tmp2[0].[14];
   		Simon_Rotate_Result[0].[14]:=Simon_tmp2[0].[13];
   		Simon_Rotate_Result[0].[13]:=Simon_tmp2[0].[12];
   		Simon_Rotate_Result[0].[12]:=Simon_tmp2[0].[11];
   		Simon_Rotate_Result[0].[11]:=Simon_tmp2[0].[10];
   		Simon_Rotate_Result[0].[10]:=Simon_tmp2[0].[9];
   		Simon_Rotate_Result[0].[9]:=Simon_tmp2[0].[8];
   		Simon_Rotate_Result[0].[8]:=Simon_tmp2[0].[7];
   		Simon_Rotate_Result[0].[7]:=Simon_tmp2[0].[6];
   		Simon_Rotate_Result[0].[6]:=Simon_tmp2[0].[5];
   		Simon_Rotate_Result[0].[5]:=Simon_tmp2[0].[4];
   		Simon_Rotate_Result[0].[4]:=Simon_tmp2[0].[3];
   		Simon_Rotate_Result[0].[3]:=Simon_tmp2[0].[2];
   		Simon_Rotate_Result[0].[2]:=Simon_tmp2[0].[1];
   		Simon_Rotate_Result[0].[1]:=Simon_tmp2[0].[0];
   	1,2:
   		Simon_Rotate_Result[0].[0]:=Simon_tmp2[0].[31];
   		Simon_Rotate_Result[0].[31]:=Simon_tmp2[0].[30];
   		Simon_Rotate_Result[0].[30]:=Simon_tmp2[0].[29];
   		Simon_Rotate_Result[0].[29]:=Simon_tmp2[0].[28];
   		Simon_Rotate_Result[0].[28]:=Simon_tmp2[0].[27];
   		Simon_Rotate_Result[0].[27]:=Simon_tmp2[0].[26];
   		Simon_Rotate_Result[0].[26]:=Simon_tmp2[0].[25];
   		Simon_Rotate_Result[0].[25]:=Simon_tmp2[0].[24];
   		Simon_Rotate_Result[0].[24]:=Simon_tmp2[0].[23];
   		Simon_Rotate_Result[0].[23]:=Simon_tmp2[0].[22];
   		Simon_Rotate_Result[0].[22]:=Simon_tmp2[0].[21];
   		Simon_Rotate_Result[0].[21]:=Simon_tmp2[0].[20];
   		Simon_Rotate_Result[0].[20]:=Simon_tmp2[0].[19];
   		Simon_Rotate_Result[0].[19]:=Simon_tmp2[0].[18];
   		Simon_Rotate_Result[0].[18]:=Simon_tmp2[0].[17];
   		Simon_Rotate_Result[0].[17]:=Simon_tmp2[0].[16];
   		Simon_Rotate_Result[0].[16]:=Simon_tmp2[0].[15];
   		Simon_Rotate_Result[0].[15]:=Simon_tmp2[0].[14];
   		Simon_Rotate_Result[0].[14]:=Simon_tmp2[0].[13];
   		Simon_Rotate_Result[0].[13]:=Simon_tmp2[0].[12];
   		Simon_Rotate_Result[0].[12]:=Simon_tmp2[0].[11];
   		Simon_Rotate_Result[0].[11]:=Simon_tmp2[0].[10];
   		Simon_Rotate_Result[0].[10]:=Simon_tmp2[0].[9];
   		Simon_Rotate_Result[0].[9]:=Simon_tmp2[0].[8];
   		Simon_Rotate_Result[0].[8]:=Simon_tmp2[0].[7];
   		Simon_Rotate_Result[0].[7]:=Simon_tmp2[0].[6];
   		Simon_Rotate_Result[0].[6]:=Simon_tmp2[0].[5];
   		Simon_Rotate_Result[0].[5]:=Simon_tmp2[0].[4];
   		Simon_Rotate_Result[0].[4]:=Simon_tmp2[0].[3];
   		Simon_Rotate_Result[0].[3]:=Simon_tmp2[0].[2];
   		Simon_Rotate_Result[0].[2]:=Simon_tmp2[0].[1];
   		Simon_Rotate_Result[0].[1]:=Simon_tmp2[0].[0];
   	3,4,5:
   		Simon_Rotate_Result[0].[0]:=Simon_tmp2[1].[31];
   		Simon_Rotate_Result[1].[31]:=Simon_tmp2[1].[30];
   		Simon_Rotate_Result[1].[30]:=Simon_tmp2[1].[29];
   		Simon_Rotate_Result[1].[29]:=Simon_tmp2[1].[28];
   		Simon_Rotate_Result[1].[28]:=Simon_tmp2[1].[27];
   		Simon_Rotate_Result[1].[27]:=Simon_tmp2[1].[26];
   		Simon_Rotate_Result[1].[26]:=Simon_tmp2[1].[25];
   		Simon_Rotate_Result[1].[25]:=Simon_tmp2[1].[24];
   		Simon_Rotate_Result[1].[24]:=Simon_tmp2[1].[23];
   		Simon_Rotate_Result[1].[23]:=Simon_tmp2[1].[22];
   		Simon_Rotate_Result[1].[22]:=Simon_tmp2[1].[21];
   		Simon_Rotate_Result[1].[21]:=Simon_tmp2[1].[20];
   		Simon_Rotate_Result[1].[20]:=Simon_tmp2[1].[19];
   		Simon_Rotate_Result[1].[19]:=Simon_tmp2[1].[18];
   		Simon_Rotate_Result[1].[18]:=Simon_tmp2[1].[17];
   		Simon_Rotate_Result[1].[17]:=Simon_tmp2[1].[16];
   		Simon_Rotate_Result[1].[16]:=Simon_tmp2[1].[15];
   		Simon_Rotate_Result[1].[15]:=Simon_tmp2[1].[14];
   		Simon_Rotate_Result[1].[14]:=Simon_tmp2[1].[13];
   		Simon_Rotate_Result[1].[13]:=Simon_tmp2[1].[12];
   		Simon_Rotate_Result[1].[12]:=Simon_tmp2[1].[11];
   		Simon_Rotate_Result[1].[11]:=Simon_tmp2[1].[10];
   		Simon_Rotate_Result[1].[10]:=Simon_tmp2[1].[9];
   		Simon_Rotate_Result[1].[9]:=Simon_tmp2[1].[8];
   		Simon_Rotate_Result[1].[8]:=Simon_tmp2[1].[7];
   		Simon_Rotate_Result[1].[7]:=Simon_tmp2[1].[6];
   		Simon_Rotate_Result[1].[6]:=Simon_tmp2[1].[5];
   		Simon_Rotate_Result[1].[5]:=Simon_tmp2[1].[4];
   		Simon_Rotate_Result[1].[4]:=Simon_tmp2[1].[3];
   		Simon_Rotate_Result[1].[3]:=Simon_tmp2[1].[2];
   		Simon_Rotate_Result[1].[2]:=Simon_tmp2[1].[1];
   		Simon_Rotate_Result[1].[1]:=Simon_tmp2[1].[0];
   		Simon_Rotate_Result[1].[0]:=Simon_tmp2[0].[31];
   		Simon_Rotate_Result[0].[31]:=Simon_tmp2[0].[30];
   		Simon_Rotate_Result[0].[30]:=Simon_tmp2[0].[29];
   		Simon_Rotate_Result[0].[29]:=Simon_tmp2[0].[28];
   		Simon_Rotate_Result[0].[28]:=Simon_tmp2[0].[27];
   		Simon_Rotate_Result[0].[27]:=Simon_tmp2[0].[26];
   		Simon_Rotate_Result[0].[26]:=Simon_tmp2[0].[25];
   		Simon_Rotate_Result[0].[25]:=Simon_tmp2[0].[24];
   		Simon_Rotate_Result[0].[24]:=Simon_tmp2[0].[23];
   		Simon_Rotate_Result[0].[23]:=Simon_tmp2[0].[22];
   		Simon_Rotate_Result[0].[22]:=Simon_tmp2[0].[21];
   		Simon_Rotate_Result[0].[21]:=Simon_tmp2[0].[20];
   		Simon_Rotate_Result[0].[20]:=Simon_tmp2[0].[19];
   		Simon_Rotate_Result[0].[19]:=Simon_tmp2[0].[18];
   		Simon_Rotate_Result[0].[18]:=Simon_tmp2[0].[17];
   		Simon_Rotate_Result[0].[17]:=Simon_tmp2[0].[16];
   		Simon_Rotate_Result[0].[16]:=Simon_tmp2[0].[15];
   		Simon_Rotate_Result[0].[15]:=Simon_tmp2[0].[14];
   		Simon_Rotate_Result[0].[14]:=Simon_tmp2[0].[13];
   		Simon_Rotate_Result[0].[13]:=Simon_tmp2[0].[12];
   		Simon_Rotate_Result[0].[12]:=Simon_tmp2[0].[11];
   		Simon_Rotate_Result[0].[11]:=Simon_tmp2[0].[10];
   		Simon_Rotate_Result[0].[10]:=Simon_tmp2[0].[9];
   		Simon_Rotate_Result[0].[9]:=Simon_tmp2[0].[8];
   		Simon_Rotate_Result[0].[8]:=Simon_tmp2[0].[7];
   		Simon_Rotate_Result[0].[7]:=Simon_tmp2[0].[6];
   		Simon_Rotate_Result[0].[6]:=Simon_tmp2[0].[5];
   		Simon_Rotate_Result[0].[5]:=Simon_tmp2[0].[4];
   		Simon_Rotate_Result[0].[4]:=Simon_tmp2[0].[3];
   		Simon_Rotate_Result[0].[3]:=Simon_tmp2[0].[2];
   		Simon_Rotate_Result[0].[2]:=Simon_tmp2[0].[1];
   		Simon_Rotate_Result[0].[1]:=Simon_tmp2[0].[0];
   End_CASE;
   
END_ROUTINE

ROUTINE SIMON_Rotate_Left2   (* structured text *)
   CASE Simon_Ver Of
   	0:
   		Simon_Rotate_Result[0].[1]:=Simon_Ciphertext[0,0].[15];
   		Simon_Rotate_Result[0].[0]:=Simon_Ciphertext[0,0].[14];
   		Simon_Rotate_Result[0].[15]:=Simon_Ciphertext[0,0].[13];
   		Simon_Rotate_Result[0].[14]:=Simon_Ciphertext[0,0].[12];
   		Simon_Rotate_Result[0].[13]:=Simon_Ciphertext[0,0].[11];
   		Simon_Rotate_Result[0].[12]:=Simon_Ciphertext[0,0].[10];
   		Simon_Rotate_Result[0].[11]:=Simon_Ciphertext[0,0].[9];
   		Simon_Rotate_Result[0].[10]:=Simon_Ciphertext[0,0].[8];
   		Simon_Rotate_Result[0].[9]:=Simon_Ciphertext[0,0].[7];
   		Simon_Rotate_Result[0].[8]:=Simon_Ciphertext[0,0].[6];
   		Simon_Rotate_Result[0].[7]:=Simon_Ciphertext[0,0].[5];
   		Simon_Rotate_Result[0].[6]:=Simon_Ciphertext[0,0].[4];
   		Simon_Rotate_Result[0].[5]:=Simon_Ciphertext[0,0].[3];
   		Simon_Rotate_Result[0].[4]:=Simon_Ciphertext[0,0].[2];
   		Simon_Rotate_Result[0].[3]:=Simon_Ciphertext[0,0].[1];
   		Simon_Rotate_Result[0].[2]:=Simon_Ciphertext[0,0].[0];
   	1,2:
   		Simon_Rotate_Result[0].[1]:=Simon_tmp2[0].[31];
   		Simon_Rotate_Result[0].[0]:=Simon_tmp2[0].[30];
   		Simon_Rotate_Result[0].[31]:=Simon_tmp2[0].[29];
   		Simon_Rotate_Result[0].[30]:=Simon_tmp2[0].[28];
   		Simon_Rotate_Result[0].[29]:=Simon_tmp2[0].[27];
   		Simon_Rotate_Result[0].[28]:=Simon_tmp2[0].[26];
   		Simon_Rotate_Result[0].[27]:=Simon_tmp2[0].[25];
   		Simon_Rotate_Result[0].[26]:=Simon_tmp2[0].[24];
   		Simon_Rotate_Result[0].[25]:=Simon_tmp2[0].[23];
   		Simon_Rotate_Result[0].[24]:=Simon_tmp2[0].[22];
   		Simon_Rotate_Result[0].[23]:=Simon_tmp2[0].[21];
   		Simon_Rotate_Result[0].[22]:=Simon_tmp2[0].[20];
   		Simon_Rotate_Result[0].[21]:=Simon_tmp2[0].[19];
   		Simon_Rotate_Result[0].[20]:=Simon_tmp2[0].[18];
   		Simon_Rotate_Result[0].[19]:=Simon_tmp2[0].[17];
   		Simon_Rotate_Result[0].[18]:=Simon_tmp2[0].[16];
   		Simon_Rotate_Result[0].[17]:=Simon_tmp2[0].[15];
   		Simon_Rotate_Result[0].[16]:=Simon_tmp2[0].[14];
   		Simon_Rotate_Result[0].[15]:=Simon_tmp2[0].[13];
   		Simon_Rotate_Result[0].[14]:=Simon_tmp2[0].[12];
   		Simon_Rotate_Result[0].[13]:=Simon_tmp2[0].[11];
   		Simon_Rotate_Result[0].[12]:=Simon_tmp2[0].[10];
   		Simon_Rotate_Result[0].[11]:=Simon_tmp2[0].[9];
   		Simon_Rotate_Result[0].[10]:=Simon_tmp2[0].[8];
   		Simon_Rotate_Result[0].[9]:=Simon_tmp2[0].[7];
   		Simon_Rotate_Result[0].[8]:=Simon_tmp2[0].[6];
   		Simon_Rotate_Result[0].[7]:=Simon_tmp2[0].[5];
   		Simon_Rotate_Result[0].[6]:=Simon_tmp2[0].[4];
   		Simon_Rotate_Result[0].[5]:=Simon_tmp2[0].[3];
   		Simon_Rotate_Result[0].[4]:=Simon_tmp2[0].[2];
   		Simon_Rotate_Result[0].[3]:=Simon_tmp2[0].[1];
   		Simon_Rotate_Result[0].[2]:=Simon_tmp2[0].[0];
   	3,4,5:
   		Simon_Rotate_Result[0].[1]:=Simon_tmp2[1].[31];
   		Simon_Rotate_Result[0].[0]:=Simon_tmp2[1].[30];
   		Simon_Rotate_Result[1].[31]:=Simon_tmp2[1].[29];
   		Simon_Rotate_Result[1].[30]:=Simon_tmp2[1].[28];
   		Simon_Rotate_Result[1].[29]:=Simon_tmp2[1].[27];
   		Simon_Rotate_Result[1].[28]:=Simon_tmp2[1].[26];
   		Simon_Rotate_Result[1].[27]:=Simon_tmp2[1].[25];
   		Simon_Rotate_Result[1].[26]:=Simon_tmp2[1].[24];
   		Simon_Rotate_Result[1].[25]:=Simon_tmp2[1].[23];
   		Simon_Rotate_Result[1].[24]:=Simon_tmp2[1].[22];
   		Simon_Rotate_Result[1].[23]:=Simon_tmp2[1].[21];
   		Simon_Rotate_Result[1].[22]:=Simon_tmp2[1].[20];
   		Simon_Rotate_Result[1].[21]:=Simon_tmp2[1].[19];
   		Simon_Rotate_Result[1].[20]:=Simon_tmp2[1].[18];
   		Simon_Rotate_Result[1].[19]:=Simon_tmp2[1].[17];
   		Simon_Rotate_Result[1].[18]:=Simon_tmp2[1].[16];
   		Simon_Rotate_Result[1].[17]:=Simon_tmp2[1].[15];
   		Simon_Rotate_Result[1].[16]:=Simon_tmp2[1].[14];
   		Simon_Rotate_Result[1].[15]:=Simon_tmp2[1].[13];
   		Simon_Rotate_Result[1].[14]:=Simon_tmp2[1].[12];
   		Simon_Rotate_Result[1].[13]:=Simon_tmp2[1].[11];
   		Simon_Rotate_Result[1].[12]:=Simon_tmp2[1].[10];
   		Simon_Rotate_Result[1].[11]:=Simon_tmp2[1].[9];
   		Simon_Rotate_Result[1].[10]:=Simon_tmp2[1].[8];
   		Simon_Rotate_Result[1].[9]:=Simon_tmp2[1].[7];
   		Simon_Rotate_Result[1].[8]:=Simon_tmp2[1].[6];
   		Simon_Rotate_Result[1].[7]:=Simon_tmp2[1].[5];
   		Simon_Rotate_Result[1].[6]:=Simon_tmp2[1].[4];
   		Simon_Rotate_Result[1].[5]:=Simon_tmp2[1].[3];
   		Simon_Rotate_Result[1].[4]:=Simon_tmp2[1].[2];
   		Simon_Rotate_Result[1].[3]:=Simon_tmp2[1].[1];
   		Simon_Rotate_Result[1].[2]:=Simon_tmp2[1].[0];
   		Simon_Rotate_Result[1].[1]:=Simon_tmp2[0].[31];
   		Simon_Rotate_Result[1].[0]:=Simon_tmp2[0].[30];
   		Simon_Rotate_Result[0].[31]:=Simon_tmp2[0].[29];
   		Simon_Rotate_Result[0].[30]:=Simon_tmp2[0].[28];
   		Simon_Rotate_Result[0].[29]:=Simon_tmp2[0].[27];
   		Simon_Rotate_Result[0].[28]:=Simon_tmp2[0].[26];
   		Simon_Rotate_Result[0].[27]:=Simon_tmp2[0].[25];
   		Simon_Rotate_Result[0].[26]:=Simon_tmp2[0].[24];
   		Simon_Rotate_Result[0].[25]:=Simon_tmp2[0].[23];
   		Simon_Rotate_Result[0].[24]:=Simon_tmp2[0].[22];
   		Simon_Rotate_Result[0].[23]:=Simon_tmp2[0].[21];
   		Simon_Rotate_Result[0].[22]:=Simon_tmp2[0].[20];
   		Simon_Rotate_Result[0].[21]:=Simon_tmp2[0].[19];
   		Simon_Rotate_Result[0].[20]:=Simon_tmp2[0].[18];
   		Simon_Rotate_Result[0].[19]:=Simon_tmp2[0].[17];
   		Simon_Rotate_Result[0].[18]:=Simon_tmp2[0].[16];
   		Simon_Rotate_Result[0].[17]:=Simon_tmp2[0].[15];
   		Simon_Rotate_Result[0].[16]:=Simon_tmp2[0].[14];
   		Simon_Rotate_Result[0].[15]:=Simon_tmp2[0].[13];
   		Simon_Rotate_Result[0].[14]:=Simon_tmp2[0].[12];
   		Simon_Rotate_Result[0].[13]:=Simon_tmp2[0].[11];
   		Simon_Rotate_Result[0].[12]:=Simon_tmp2[0].[10];
   		Simon_Rotate_Result[0].[11]:=Simon_tmp2[0].[9];
   		Simon_Rotate_Result[0].[10]:=Simon_tmp2[0].[8];
   		Simon_Rotate_Result[0].[9]:=Simon_tmp2[0].[7];
   		Simon_Rotate_Result[0].[8]:=Simon_tmp2[0].[6];
   		Simon_Rotate_Result[0].[7]:=Simon_tmp2[0].[5];
   		Simon_Rotate_Result[0].[6]:=Simon_tmp2[0].[4];
   		Simon_Rotate_Result[0].[5]:=Simon_tmp2[0].[3];
   		Simon_Rotate_Result[0].[4]:=Simon_tmp2[0].[2];
   		Simon_Rotate_Result[0].[3]:=Simon_tmp2[0].[1];
   		Simon_Rotate_Result[0].[2]:=Simon_tmp2[0].[0];
   End_CASE;
   
END_ROUTINE

ROUTINE SIMON_Rotate_Left8   (* structured text *)
   CASE Simon_Ver Of
   	0:
   		Simon_Rotate_Result[0].[7]:=Simon_Ciphertext[0,0].[15];
   		Simon_Rotate_Result[0].[6]:=Simon_Ciphertext[0,0].[14];
   		Simon_Rotate_Result[0].[5]:=Simon_Ciphertext[0,0].[13];
   		Simon_Rotate_Result[0].[4]:=Simon_Ciphertext[0,0].[12];
   		Simon_Rotate_Result[0].[3]:=Simon_Ciphertext[0,0].[11];
   		Simon_Rotate_Result[0].[2]:=Simon_Ciphertext[0,0].[10];
   		Simon_Rotate_Result[0].[1]:=Simon_Ciphertext[0,0].[9];
   		Simon_Rotate_Result[0].[0]:=Simon_Ciphertext[0,0].[8];
   		Simon_Rotate_Result[0].[15]:=Simon_Ciphertext[0,0].[7];
   		Simon_Rotate_Result[0].[14]:=Simon_Ciphertext[0,0].[6];
   		Simon_Rotate_Result[0].[13]:=Simon_Ciphertext[0,0].[5];
   		Simon_Rotate_Result[0].[12]:=Simon_Ciphertext[0,0].[4];
   		Simon_Rotate_Result[0].[11]:=Simon_Ciphertext[0,0].[3];
   		Simon_Rotate_Result[0].[10]:=Simon_Ciphertext[0,0].[2];
   		Simon_Rotate_Result[0].[9]:=Simon_Ciphertext[0,0].[1];
   		Simon_Rotate_Result[0].[8]:=Simon_Ciphertext[0,0].[0];
   	1,2:
   		Simon_Rotate_Result[0].[7]:=Simon_tmp2[0].[31];
   		Simon_Rotate_Result[0].[6]:=Simon_tmp2[0].[30];
   		Simon_Rotate_Result[0].[5]:=Simon_tmp2[0].[29];
   		Simon_Rotate_Result[0].[4]:=Simon_tmp2[0].[28];
   		Simon_Rotate_Result[0].[3]:=Simon_tmp2[0].[27];
   		Simon_Rotate_Result[0].[2]:=Simon_tmp2[0].[26];
   		Simon_Rotate_Result[0].[1]:=Simon_tmp2[0].[25];
   		Simon_Rotate_Result[0].[0]:=Simon_tmp2[0].[24];
   		Simon_Rotate_Result[0].[31]:=Simon_tmp2[0].[23];
   		Simon_Rotate_Result[0].[30]:=Simon_tmp2[0].[22];
   		Simon_Rotate_Result[0].[29]:=Simon_tmp2[0].[21];
   		Simon_Rotate_Result[0].[28]:=Simon_tmp2[0].[20];
   		Simon_Rotate_Result[0].[27]:=Simon_tmp2[0].[19];
   		Simon_Rotate_Result[0].[26]:=Simon_tmp2[0].[18];
   		Simon_Rotate_Result[0].[25]:=Simon_tmp2[0].[17];
   		Simon_Rotate_Result[0].[24]:=Simon_tmp2[0].[16];
   		Simon_Rotate_Result[0].[23]:=Simon_tmp2[0].[15];
   		Simon_Rotate_Result[0].[22]:=Simon_tmp2[0].[14];
   		Simon_Rotate_Result[0].[21]:=Simon_tmp2[0].[13];
   		Simon_Rotate_Result[0].[20]:=Simon_tmp2[0].[12];
   		Simon_Rotate_Result[0].[19]:=Simon_tmp2[0].[11];
   		Simon_Rotate_Result[0].[18]:=Simon_tmp2[0].[10];
   		Simon_Rotate_Result[0].[17]:=Simon_tmp2[0].[9];
   		Simon_Rotate_Result[0].[16]:=Simon_tmp2[0].[8];
   		Simon_Rotate_Result[0].[15]:=Simon_tmp2[0].[7];
   		Simon_Rotate_Result[0].[14]:=Simon_tmp2[0].[6];
   		Simon_Rotate_Result[0].[13]:=Simon_tmp2[0].[5];
   		Simon_Rotate_Result[0].[12]:=Simon_tmp2[0].[4];
   		Simon_Rotate_Result[0].[11]:=Simon_tmp2[0].[3];
   		Simon_Rotate_Result[0].[10]:=Simon_tmp2[0].[2];
   		Simon_Rotate_Result[0].[9]:=Simon_tmp2[0].[1];
   		Simon_Rotate_Result[0].[8]:=Simon_tmp2[0].[0];
   	3,4,5:
   		Simon_Rotate_Result[0].[7]:=Simon_tmp2[1].[31];
   		Simon_Rotate_Result[0].[6]:=Simon_tmp2[1].[30];
   		Simon_Rotate_Result[0].[5]:=Simon_tmp2[1].[29];
   		Simon_Rotate_Result[0].[4]:=Simon_tmp2[1].[28];
   		Simon_Rotate_Result[0].[3]:=Simon_tmp2[1].[27];
   		Simon_Rotate_Result[0].[2]:=Simon_tmp2[1].[26];
   		Simon_Rotate_Result[0].[1]:=Simon_tmp2[1].[25];
   		Simon_Rotate_Result[0].[0]:=Simon_tmp2[1].[24];
   		Simon_Rotate_Result[1].[31]:=Simon_tmp2[1].[23];
   		Simon_Rotate_Result[1].[30]:=Simon_tmp2[1].[22];
   		Simon_Rotate_Result[1].[29]:=Simon_tmp2[1].[21];
   		Simon_Rotate_Result[1].[28]:=Simon_tmp2[1].[20];
   		Simon_Rotate_Result[1].[27]:=Simon_tmp2[1].[19];
   		Simon_Rotate_Result[1].[26]:=Simon_tmp2[1].[18];
   		Simon_Rotate_Result[1].[25]:=Simon_tmp2[1].[17];
   		Simon_Rotate_Result[1].[24]:=Simon_tmp2[1].[16];
   		Simon_Rotate_Result[1].[23]:=Simon_tmp2[1].[15];
   		Simon_Rotate_Result[1].[22]:=Simon_tmp2[1].[14];
   		Simon_Rotate_Result[1].[21]:=Simon_tmp2[1].[13];
   		Simon_Rotate_Result[1].[20]:=Simon_tmp2[1].[12];
   		Simon_Rotate_Result[1].[19]:=Simon_tmp2[1].[11];
   		Simon_Rotate_Result[1].[18]:=Simon_tmp2[1].[10];
   		Simon_Rotate_Result[1].[17]:=Simon_tmp2[1].[9];
   		Simon_Rotate_Result[1].[16]:=Simon_tmp2[1].[8];
   		Simon_Rotate_Result[1].[15]:=Simon_tmp2[1].[7];
   		Simon_Rotate_Result[1].[14]:=Simon_tmp2[1].[6];
   		Simon_Rotate_Result[1].[13]:=Simon_tmp2[1].[5];
   		Simon_Rotate_Result[1].[12]:=Simon_tmp2[1].[4];
   		Simon_Rotate_Result[1].[11]:=Simon_tmp2[1].[3];
   		Simon_Rotate_Result[1].[10]:=Simon_tmp2[1].[2];
   		Simon_Rotate_Result[1].[9]:=Simon_tmp2[1].[1];
   		Simon_Rotate_Result[1].[8]:=Simon_tmp2[1].[0];
   		Simon_Rotate_Result[1].[7]:=Simon_tmp2[0].[31];
   		Simon_Rotate_Result[1].[6]:=Simon_tmp2[0].[30];
   		Simon_Rotate_Result[1].[5]:=Simon_tmp2[0].[29];
   		Simon_Rotate_Result[1].[4]:=Simon_tmp2[0].[28];
   		Simon_Rotate_Result[1].[3]:=Simon_tmp2[0].[27];
   		Simon_Rotate_Result[1].[2]:=Simon_tmp2[0].[26];
   		Simon_Rotate_Result[1].[1]:=Simon_tmp2[0].[25];
   		Simon_Rotate_Result[1].[0]:=Simon_tmp2[0].[24];
   		Simon_Rotate_Result[0].[31]:=Simon_tmp2[0].[23];
   		Simon_Rotate_Result[0].[30]:=Simon_tmp2[0].[22];
   		Simon_Rotate_Result[0].[29]:=Simon_tmp2[0].[21];
   		Simon_Rotate_Result[0].[28]:=Simon_tmp2[0].[20];
   		Simon_Rotate_Result[0].[27]:=Simon_tmp2[0].[19];
   		Simon_Rotate_Result[0].[26]:=Simon_tmp2[0].[18];
   		Simon_Rotate_Result[0].[25]:=Simon_tmp2[0].[17];
   		Simon_Rotate_Result[0].[24]:=Simon_tmp2[0].[16];
   		Simon_Rotate_Result[0].[23]:=Simon_tmp2[0].[15];
   		Simon_Rotate_Result[0].[22]:=Simon_tmp2[0].[14];
   		Simon_Rotate_Result[0].[21]:=Simon_tmp2[0].[13];
   		Simon_Rotate_Result[0].[20]:=Simon_tmp2[0].[12];
   		Simon_Rotate_Result[0].[19]:=Simon_tmp2[0].[11];
   		Simon_Rotate_Result[0].[18]:=Simon_tmp2[0].[10];
   		Simon_Rotate_Result[0].[17]:=Simon_tmp2[0].[9];
   		Simon_Rotate_Result[0].[16]:=Simon_tmp2[0].[8];
   		Simon_Rotate_Result[0].[15]:=Simon_tmp2[0].[7];
   		Simon_Rotate_Result[0].[14]:=Simon_tmp2[0].[6];
   		Simon_Rotate_Result[0].[13]:=Simon_tmp2[0].[5];
   		Simon_Rotate_Result[0].[12]:=Simon_tmp2[0].[4];
   		Simon_Rotate_Result[0].[11]:=Simon_tmp2[0].[3];
   		Simon_Rotate_Result[0].[10]:=Simon_tmp2[0].[2];
   		Simon_Rotate_Result[0].[9]:=Simon_tmp2[0].[1];
   		Simon_Rotate_Result[0].[8]:=Simon_tmp2[0].[0];
   End_CASE;
   
END_ROUTINE
END_PROGRAM
